// TwinCAT 3 PLC project Untitled1
// ProgramVersion: 3.1.4024.0
// libraries:
//   Tc2_Standard, * (Beckhoff Automation GmbH)
//   Tc2_System, * (Beckhoff Automation GmbH)
//   Tc3_Module, * (Beckhoff Automation GmbH)
//   VisuSymbols,3.5.10.0,System
// project tree:
//   / GlobalTextList.TcGTLO, PlcTask.TcTTO, task1.TcTTO, task2.TcTTO, task3.TcTTO, Task_4.TcTTO, Visualization Manager.TcVMO (not stored), Visualization.TcVIS
//   GVLs/ GVL.TcGVL
//   POUs/ Main.TcPOU, PRG_BeerSession.TcPOU, PRG_GameSession.TcPOU, PRG_TrainTrip.TcPOU
// real-time tasks:
//   TASK PlcTask: cycle T#10ms, priority 20, ADS port 350
//   TASK Task 4: cycle T#10ms, priority 1, ADS port 351
//   TASK task1: cycle T#10ms, priority 21, ADS port 352
//   TASK task2: cycle T#10ms, priority 22, ADS port 353
//   TASK task3: cycle T#10ms, priority 23, ADS port 354

CONFIGURATION Untitled1
    RESOURCE PLC ON TwinCAT3
        TASK PlcTask(INTERVAL := T#10ms, PRIORITY := 20);
        TASK task1(INTERVAL := T#10ms, PRIORITY := 21);
        TASK task2(INTERVAL := T#10ms, PRIORITY := 22);
        TASK task3(INTERVAL := T#10ms, PRIORITY := 23);
        TASK Task_4(INTERVAL := T#10ms, PRIORITY := 1);
        PROGRAM PRG_TrainTrip WITH task1 : PRG_TrainTrip;
        PROGRAM PRG_BeerSession WITH task2 : PRG_BeerSession;
        PROGRAM PRG_GameSession WITH task3 : PRG_GameSession;
        PROGRAM Main WITH Task_4 : Main;
    END_RESOURCE
END_CONFIGURATION

// ---- GVLs/GVL.TcGVL
VAR_GLOBAL
    (* Treinreis *)
    ReisGestart      : BOOL := FALSE;
    OverstapBereikt  : BOOL := FALSE;
    Aangekomen       : BOOL := FALSE;

    (* Bier *)
    Biertjes         : UINT := 0;

    (* Spel *)
    SpelGestart      : BOOL := FALSE;
    Ronde            : UINT := 0;

    (* Avond *)
    AvondKlaar       : BOOL := FALSE;
END_VAR

// ---- POUs/PRG_TrainTrip.TcPOU
PROGRAM PRG_TrainTrip
VAR
    T_Overstap : TON;
    T_Aankomst : TON;
END_VAR

IF NOT ReisGestart THEN
    ReisGestart := TRUE;
END_IF

(* Trein naar overstap *)
IF ReisGestart AND NOT OverstapBereikt THEN
    T_Overstap(IN := TRUE, PT := T#5S);

    IF T_Overstap.Q THEN
        OverstapBereikt := TRUE;
        T_Overstap(IN := FALSE);
    END_IF
END_IF

(* Trein naar eindbestemming *)
IF OverstapBereikt AND NOT Aangekomen THEN
    T_Aankomst(IN := TRUE, PT := T#5S);

    IF T_Aankomst.Q THEN
        Aangekomen := TRUE;
        T_Aankomst(IN := FALSE);
    END_IF
END_IF

END_PROGRAM

// ---- POUs/PRG_BeerSession.TcPOU
PROGRAM PRG_BeerSession
VAR
    T_Biertje : TON;
END_VAR

IF Aangekomen AND NOT AvondKlaar THEN
    IF Biertjes < 5 THEN
        T_Biertje(IN := TRUE, PT := T#4S);

        IF T_Biertje.Q THEN
            Biertjes := Biertjes + 1;
            T_Biertje(IN := FALSE);
        END_IF
    END_IF
END_IF

END_PROGRAM

// ---- POUs/PRG_GameSession.TcPOU
PROGRAM PRG_GameSession
VAR
    T_Ronde : TON;
END_VAR

IF (Biertjes >= 3) AND NOT SpelGestart THEN
    SpelGestart := TRUE;
END_IF

IF SpelGestart AND (Ronde < 10) THEN
    T_Ronde(IN := TRUE, PT := T#4S);

    IF T_Ronde.Q THEN
        Ronde := Ronde + 1;
        T_Ronde(IN := FALSE);
    END_IF
END_IF

IF Ronde >= 10 THEN
    AvondKlaar := TRUE;
END_IF

END_PROGRAM

// ---- POUs/Main.TcPOU
PROGRAM Main
VAR
    KlaarVoorBier : BOOL;
    KlaarVoorSpel : BOOL;
END_VAR


KlaarVoorBier := Aangekomen;
KlaarVoorSpel := (Biertjes >= 3);

END_PROGRAM

// ---- Visualization.TcVIS
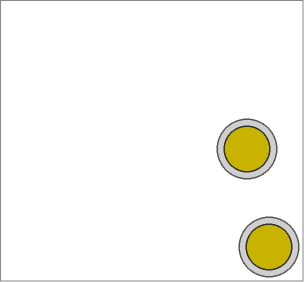
VISUALIZATION Visualization  // 304x282
    Lamp1 (212,114 70x70), variable: Main.KlaarVoorBier, style: Lamp-Lamp1-Yellow
    Lamp1 (234,212 70x70), variable: Main.KlaarVoorSpel, style: Lamp-Lamp1-Yellow
END_VISUALIZATION
